DATA_BLOCK "Data_block_20"
{ S7_Optimized_Access := 'FALSE' }
VERSION : 0.1
NON_RETAIN
   VAR
      S7Tag0 : Word;
      S7Tag1 : Word;
      S7Tag2 : Word;
      S7Tag3 : Word;
      S7Tag4 : Word;
      S7Tag5 : Word;
      S7Tag6 : Word;
      S7Tag7 : Word;
      S7Tag8 : Word;
      S7Tag9 : Word;
      S7Tag10 : Word;
      S7Tag11 : Word;
      S7Tag12 : Word;
      S7Tag13 : Word;
      S7Tag14 : Word;
      S7Tag15 : Word;
      S7Tag16 : Word;
      S7Tag17 : Word;
      S7Tag18 : Word;
      S7Tag19 : Word;
      S7Tag20 : Word;
      S7Tag21 : Word;
      S7Tag22 : Word;
      S7Tag23 : Word;
      S7Tag24 : Word;
      S7Tag25 : Word;
      S7Tag26 : Word;
      S7Tag27 : Word;
      S7Tag28 : Word;
      S7Tag29 : Word;
      S7Tag30 : Word;
      S7Tag31 : Word;
      S7Tag32 : Word;
      S7Tag33 : Word;
      S7Tag34 : Word;
      S7Tag35 : Word;
      S7Tag36 : Word;
      S7Tag37 : Word;
      S7Tag38 : Word;
      S7Tag39 : Word;
      S7Tag40 : Word;
      S7Tag41 : Word;
      S7Tag42 : Word;
      S7Tag43 : Word;
      S7Tag44 : Word;
      S7Tag45 : Word;
      S7Tag46 : Word;
      S7Tag47 : Word;
      S7Tag48 : Word;
      S7Tag49 : Word;
      S7Tag50 : Word;
      S7Tag51 : Word;
      S7Tag52 : Word;
      S7Tag53 : Word;
      S7Tag54 : Word;
      S7Tag55 : Word;
      S7Tag56 : Word;
      S7Tag57 : Word;
      S7Tag58 : Word;
      S7Tag59 : Word;
      S7Tag60 : Word;
      S7Tag61 : Word;
      S7Tag62 : Word;
      S7Tag63 : Word;
      S7Tag64 : Word;
      S7Tag65 : Word;
      S7Tag66 : Word;
      S7Tag67 : Word;
      S7Tag68 : Word;
      S7Tag69 : Word;
      S7Tag70 : Word;
      S7Tag71 : Word;
      S7Tag72 : Word;
      S7Tag73 : Word;
      S7Tag74 : Word;
      S7Tag75 : Word;
      S7Tag76 : Word;
      S7Tag77 : Word;
      S7Tag78 : Word;
      S7Tag79 : Word;
      S7Tag80 : Word;
      S7Tag81 : Word;
      S7Tag82 : Word;
      S7Tag83 : Word;
      S7Tag84 : Word;
      S7Tag85 : Word;
      S7Tag86 : Word;
      S7Tag87 : Word;
      S7Tag88 : Word;
      S7Tag89 : Word;
      S7Tag90 : Word;
      S7Tag91 : Word;
      S7Tag92 : Word;
      S7Tag93 : Word;
      S7Tag94 : Word;
      S7Tag95 : Word;
      S7Tag96 : Word;
      S7Tag97 : Word;
      S7Tag98 : Word;
      S7Tag99 : Word;
      S7Tag100 : Word;
      S7Tag101 : Word;
      S7Tag102 : Word;
      S7Tag103 : Word;
      S7Tag104 : Word;
      S7Tag105 : Word;
      S7Tag106 : Word;
      S7Tag107 : Word;
      S7Tag108 : Word;
      S7Tag109 : Word;
      S7Tag110 : Word;
      S7Tag111 : Word;
      S7Tag112 : Word;
      S7Tag113 : Word;
      S7Tag114 : Word;
      S7Tag115 : Word;
      S7Tag116 : Word;
      S7Tag117 : Word;
      S7Tag118 : Word;
      S7Tag119 : Word;
      S7Tag120 : Word;
      S7Tag121 : Word;
      S7Tag122 : Word;
      S7Tag123 : Word;
      S7Tag124 : Word;
      S7Tag125 : Word;
      S7Tag126 : Word;
      S7Tag127 : Word;
      S7Tag128 : Word;
      S7Tag129 : Word;
      S7Tag130 : Word;
      S7Tag131 : Word;
      S7Tag132 : Word;
      S7Tag133 : Word;
      S7Tag134 : Word;
      S7Tag135 : Word;
      S7Tag136 : Word;
      S7Tag137 : Word;
      S7Tag138 : Word;
      S7Tag139 : Word;
      S7Tag140 : Word;
      S7Tag141 : Word;
      S7Tag142 : Word;
      S7Tag143 : Word;
      S7Tag144 : Word;
      S7Tag145 : Word;
      S7Tag146 : Word;
      S7Tag147 : Word;
      S7Tag148 : Word;
      S7Tag149 : Word;
      S7Tag150 : Word;
      S7Tag151 : Word;
      S7Tag152 : Word;
      S7Tag153 : Word;
      S7Tag154 : Word;
      S7Tag155 : Word;
      S7Tag156 : Word;
      S7Tag157 : Word;
      S7Tag158 : Word;
      S7Tag159 : Word;
      S7Tag160 : Word;
      S7Tag161 : Word;
      S7Tag162 : Word;
      S7Tag163 : Word;
      S7Tag164 : Word;
      S7Tag165 : Word;
      S7Tag166 : Word;
      S7Tag167 : Word;
      S7Tag168 : Word;
      S7Tag169 : Word;
      S7Tag170 : Word;
      S7Tag171 : Word;
      S7Tag172 : Word;
      S7Tag173 : Word;
      S7Tag174 : Word;
      S7Tag175 : Word;
      S7Tag176 : Word;
      S7Tag177 : Word;
      S7Tag178 : Word;
      S7Tag179 : Word;
      S7Tag180 : Word;
      S7Tag181 : Word;
      S7Tag182 : Word;
      S7Tag183 : Word;
      S7Tag184 : Word;
      S7Tag185 : Word;
      S7Tag186 : Word;
      S7Tag187 : Word;
      S7Tag188 : Word;
      S7Tag189 : Word;
      S7Tag190 : Word;
      S7Tag191 : Word;
      S7Tag192 : Word;
      S7Tag193 : Word;
      S7Tag194 : Word;
      S7Tag195 : Word;
      S7Tag196 : Word;
      S7Tag197 : Word;
      S7Tag198 : Word;
      S7Tag199 : Word;
      S7Tag200 : Word;
      S7Tag201 : Word;
      S7Tag202 : Word;
      S7Tag203 : Word;
      S7Tag204 : Word;
      S7Tag205 : Word;
      S7Tag206 : Word;
      S7Tag207 : Word;
      S7Tag208 : Word;
      S7Tag209 : Word;
      S7Tag210 : Word;
      S7Tag211 : Word;
      S7Tag212 : Word;
      S7Tag213 : Word;
      S7Tag214 : Word;
      S7Tag215 : Word;
      S7Tag216 : Word;
      S7Tag217 : Word;
      S7Tag218 : Word;
      S7Tag219 : Word;
      S7Tag220 : Word;
      S7Tag221 : Word;
      S7Tag222 : Word;
      S7Tag223 : Word;
      S7Tag224 : Word;
      S7Tag225 : Word;
      S7Tag226 : Word;
      S7Tag227 : Word;
      S7Tag228 : Word;
      S7Tag229 : Word;
      S7Tag230 : Word;
      S7Tag231 : Word;
      S7Tag232 : Word;
      S7Tag233 : Word;
      S7Tag234 : Word;
      S7Tag235 : Word;
      S7Tag236 : Word;
      S7Tag237 : Word;
      S7Tag238 : Word;
      S7Tag239 : Word;
      S7Tag240 : Word;
      S7Tag241 : Word;
      S7Tag242 : Word;
      S7Tag243 : Word;
      S7Tag244 : Word;
      S7Tag245 : Word;
      S7Tag246 : Word;
      S7Tag247 : Word;
      S7Tag248 : Word;
      S7Tag249 : Word;
      S7Tag250 : Word;
      S7Tag251 : Word;
      S7Tag252 : Word;
      S7Tag253 : Word;
      S7Tag254 : Word;
      S7Tag255 : Word;
      S7Tag256 : Word;
      S7Tag257 : Word;
      S7Tag258 : Word;
      S7Tag259 : Word;
      S7Tag260 : Word;
      S7Tag261 : Word;
      S7Tag262 : Word;
      S7Tag263 : Word;
      S7Tag264 : Word;
      S7Tag265 : Word;
      S7Tag266 : Word;
      S7Tag267 : Word;
      S7Tag268 : Word;
      S7Tag269 : Word;
      S7Tag270 : Word;
      S7Tag271 : Word;
      S7Tag272 : Word;
      S7Tag273 : Word;
      S7Tag274 : Word;
      S7Tag275 : Word;
      S7Tag276 : Word;
      S7Tag277 : Word;
      S7Tag278 : Word;
      S7Tag279 : Word;
      S7Tag280 : Word;
      S7Tag281 : Word;
      S7Tag282 : Word;
      S7Tag283 : Word;
      S7Tag284 : Word;
      S7Tag285 : Word;
      S7Tag286 : Word;
      S7Tag287 : Word;
      S7Tag288 : Word;
      S7Tag289 : Word;
      S7Tag290 : Word;
      S7Tag291 : Word;
      S7Tag292 : Word;
      S7Tag293 : Word;
      S7Tag294 : Word;
      S7Tag295 : Word;
      S7Tag296 : Word;
      S7Tag297 : Word;
      S7Tag298 : Word;
      S7Tag299 : Word;
      S7Tag300 : Word;
      S7Tag301 : Word;
      S7Tag302 : Word;
      S7Tag303 : Word;
      S7Tag304 : Word;
      S7Tag305 : Word;
      S7Tag306 : Word;
      S7Tag307 : Word;
      S7Tag308 : Word;
      S7Tag309 : Word;
      S7Tag310 : Word;
      S7Tag311 : Word;
      S7Tag312 : Word;
      S7Tag313 : Word;
      S7Tag314 : Word;
      S7Tag315 : Word;
      S7Tag316 : Word;
      S7Tag317 : Word;
      S7Tag318 : Word;
      S7Tag319 : Word;
      S7Tag320 : Word;
      S7Tag321 : Word;
      S7Tag322 : Word;
      S7Tag323 : Word;
      S7Tag324 : Word;
      S7Tag325 : Word;
      S7Tag326 : Word;
      S7Tag327 : Word;
      S7Tag328 : Word;
      S7Tag329 : Word;
      S7Tag330 : Word;
      S7Tag331 : Word;
      S7Tag332 : Word;
      S7Tag333 : Word;
      S7Tag334 : Word;
      S7Tag335 : Word;
      S7Tag336 : Word;
      S7Tag337 : Word;
      S7Tag338 : Word;
      S7Tag339 : Word;
      S7Tag340 : Word;
      S7Tag341 : Word;
      S7Tag342 : Word;
      S7Tag343 : Word;
      S7Tag344 : Word;
      S7Tag345 : Word;
      S7Tag346 : Word;
      S7Tag347 : Word;
      S7Tag348 : Word;
      S7Tag349 : Word;
      S7Tag350 : Word;
      S7Tag351 : Word;
      S7Tag352 : Word;
      S7Tag353 : Word;
      S7Tag354 : Word;
      S7Tag355 : Word;
      S7Tag356 : Word;
      S7Tag357 : Word;
      S7Tag358 : Word;
      S7Tag359 : Word;
      S7Tag360 : Word;
      S7Tag361 : Word;
      S7Tag362 : Word;
      S7Tag363 : Word;
      S7Tag364 : Word;
      S7Tag365 : Word;
      S7Tag366 : Word;
      S7Tag367 : Word;
      S7Tag368 : Word;
      S7Tag369 : Word;
      S7Tag370 : Word;
      S7Tag371 : Word;
      S7Tag372 : Word;
      S7Tag373 : Word;
      S7Tag374 : Word;
      S7Tag375 : Word;
      S7Tag376 : Word;
      S7Tag377 : Word;
      S7Tag378 : Word;
      S7Tag379 : Word;
      S7Tag380 : Word;
      S7Tag381 : Word;
      S7Tag382 : Word;
      S7Tag383 : Word;
      S7Tag384 : Word;
      S7Tag385 : Word;
      S7Tag386 : Word;
      S7Tag387 : Word;
      S7Tag388 : Word;
      S7Tag389 : Word;
      S7Tag390 : Word;
      S7Tag391 : Word;
      S7Tag392 : Word;
      S7Tag393 : Word;
      S7Tag394 : Word;
      S7Tag395 : Word;
      S7Tag396 : Word;
      S7Tag397 : Word;
      S7Tag398 : Word;
      S7Tag399 : Word;
   END_VAR


BEGIN

END_DATA_BLOCK
